// TIA Portal V17 export
// export: Created 2022-07-05T08:49:25.4389846Z, ExportSetting WithDefaults, DisplayName Totally Integrated Automation Portal, DisplayVersion V17, DisplayName TIA Portal Openness, DisplayVersion V17, DisplayName TIA Portal Version Control Interface, DisplayVersion V17, DisplayName STEP 7 Professional, DisplayVersion V17, DisplayName STEP 7 Safety, DisplayVersion V17, DisplayName WinCC Advanced, DisplayVersion V17
DATA_BLOCK "InstCounter"   // DB2
VERSION : 0.1
// stored: AutoNumber true, DBAccessibleFromOPCUA true, DBAccessibleFromWebserver true, InstanceOfName Counter, InstanceOfType FB
"Counter"
   // VAR_INPUT
   //    startCounting { ExternalWritable := 'False'} : Bool;
   //    endValue : DInt;
   //    frequency : Bool;
   // END_VAR
   // VAR_OUTPUT
   //    valueResetted { ExternalWritable := 'False'} : Bool;
   //    actValue { ExternalWritable := 'False'} : DInt;
   // END_VAR
   // VAR
   //    statValue : DInt;
   //    statEndValue : DInt;
   //    InstRTrig { S7_SetPoint := 'True'} : R_TRIG;
   //    statFreqTrig : Bool;
   // END_VAR
BEGIN
END_DATA_BLOCK
